(* Logix 5000 project; controller Test vendor 1 type 14 code 164 rev 34.11; software revision 34.01 *)
// ABC Logic

TASK MainTask (continuous, watchdog 500 ms) : MainProgram

MODULES
   Local : vendor 1 type 14 code 164 (ICP 0, rev 34.11)
      IOCARD1 : 1756-IB16 (ICP 1, rev 3.1, Input RPI 20 ms)
END_MODULES

PROGRAM MainProgram   (* main routine MainRoutine *)

ROUTINE MainRoutine   (* ladder *)
END_ROUTINE
END_PROGRAM
